(* PLC project Generated.project, CODESYS CODESYS V3.5 SP19 Patch 1 *)
(* stored: creationDateTime 2026-09-14T14:47:22.317175, modificationDateTime 2026-09-14T14:47:22.317175 *)

(* ======================================================================= 🔌 ST_ContactorCheck — Double vérification commande/retour contacteur ─────────────────────────────────────────────────────────────── 🎯 Rôle : Structure de diagnostic pour vérification commande vs retour 📊 Diagnostic : Détection des défauts contacteur (StuckClosed / StuckOpen) 📄 Doc métier : DOC/AF/AF_Partie-03_Contrats_Composants_v2.3.md §2 ======================================================================= *)
TYPE ST_ContactorCheck : STRUCT
  Command : BOOL;  (* Ordre envoyé au contacteur (TRUE = fermé/actif) *)
  Feedback : BOOL;  (* Retour d'état câblé (TRUE = effectivement fermé) *)
  StuckClosed : BOOL;  (* Diag : commande OFF mais retour ON depuis trop longtemps → PowerCutOff *)
  StuckOpen : BOOL;  (* Diag : commande ON mais retour OFF depuis trop longtemps *)
END_STRUCT;
END_TYPE

(* ======================================================================= 🧩 ST_Fault — Brique socle défaut (2 vues : live + latchée) ─────────────────────────────────────────────────────────────── 🎯 Rôle : porter l'état défaut d'un composant, applicable dans TOUS les cas (acquittable ou non), sans brique warning séparée. • Vue LIVE (Error / ErrorId) : suit la cause, retombe seule à 0. • Vue LATCHÉE (Latched / LatchedId): mémorisée au défaut, reste jusqu'au front Reset. Le choix acquittable / non-acquittable se fait PAR CAUSE (ST_FaultCause.Latching), jamais par bloc. 🔒 Sécurité : interlock TOUJOURS sur la cause brute (Error / ErrorId), jamais sur l'acquittement. Reset TOUJOURS effectif, jamais conditionné (std §9). 🧬 Composition : brique de base réutilisable — sortie de FB, struct métier, GVL. Texte IHM NON stocké ici : dérivé côté IHM depuis LatchedId / ErrorId. 📄 Doc : DOC/STDS/CODE_QUALITY_STANDARDS.md §2quinquies / §9 ======================================================================= *)
TYPE ST_Fault : STRUCT
  Error : BOOL;  (* <-- [DIAG] vue LIVE : au moins une cause présente maintenant *)
  ErrorId : WORD;  (* <-- [DIAG] bitfield des causes présentes maintenant (0 si aucune) *)
  Latched : BOOL;  (* <-- [DIAG] vue LATCHÉE : défaut non acquitté, reste jusqu'au front Reset *)
  LatchedId : WORD;  (* <-- [DIAG] ErrorId figé à l'apparition du défaut, effacé au Reset *)
END_STRUCT;
END_TYPE

(* ======================================================================= 🧩 ST_FaultCause — Cause élémentaire alimentant ST_Fault (socle FB_FaultCore) ─────────────────────────────────────────────────────────────── 🎯 Rôle : une cause exprimée EN CLAIR (BOOL + libellé), sans bitfield ni masque. Le FB métier remplit une liste (ARRAY[0..15] OF ST_FaultCause) ; le socle FB_FaultCore en déduit ST_Fault (vue live + vue latchée). 🔒 Sécurité : interlock TOUJOURS sur Active (cause brute), jamais sur le latch. Latching = TRUE → la cause ARME la vue latchée (défaut à acquitter). Latching = FALSE → la cause n'alimente que la vue live (retombe seule). Fail-safe : une cause laissée à Latching=FALSE reste visible en live — pour la rendre acquittable, il faut le déclarer explicitement. 📄 Doc : DOC/STDS/CODE_QUALITY_STANDARDS.md §2quinquies / §9 ======================================================================= *)
TYPE ST_FaultCause : STRUCT
  Active : BOOL;  (* 1 = cause présente maintenant (interlock sur cette valeur) *)
  Latching : BOOL;  (* 1 = cause à acquitter (arme Latched) ; 0 = live seulement *)
  Texte : STRING;  (* libellé prêt IHM (non stocké dans ST_Fault, dérivé côté IHM) *)
END_STRUCT;
END_TYPE

(* ======================================================================= 🪝 ST_fbWinch_Cfg — Configuration statique d'un treuil ─────────────────────────────────────────────────────────────── 🎯 Rôle : Réglages persistants propres à l'instance treuil (statique) 📄 Doc métier : DOC/AF/AF_Partie-10_Fonction_Winch_v2.1.md 📤 Producteur : configuration persistante 📥 Consommateur : FB_Winch (statique uniquement) 🔒 Structs cibles + champs conservés pour garder le décodage %→palier et les deux cadences de rampe DANS FB_Winch (comportement bit-identique). Le champ StepRampDelay est déclaré mais non consommé (usage aval). ======================================================================= *)
TYPE ST_fbWinch_Cfg : STRUCT
  SpeedStepTable : ST_SpeedStepTable;  (* === TABLE DES PALIERS === Table de seuils des paliers de vitesse *)
  DirectionInterlockDelayAscent : TIME := TIME#800ms;  (* === INTERLOCK CHANGEMENT DE SENS === Delai interlock inversion vers montee *)
  DirectionInterlockDelayDescent : TIME := TIME#500ms;  (* Delai interlock inversion vers descente *)
  StepRampDelay : TIME := TIME#700ms;  (* === CADENCE DE RAMPE PALIER === [cible] Tempo de rampe palier (usage aval) *)
  StepRampDelayAscent : TIME := TIME#700ms;  (* [08a] Cadence palier montee (D10, dedie) *)
  StepRampDelayDescent : TIME := TIME#500ms;  (* [08a] Cadence palier descending (D10, dedie) *)
  ContactorFeedbackTimeout : TIME := TIME#500ms;  (* === RETOMBÉE CONTACTEURS === Delai d'attente retombee des contacteurs *)
  SlowdownDistanceTop_M : REAL := 0.5;  (* === RALENTISSEMENT BORDURE === Distance avant limite haute pour ralentir (m) : 0 = arrêt au seuil *)
  SlowdownDistanceBottom_M : REAL := 1;  (* Distance avant limite basse pour ralentir (m) *)
  SlowdownMaxStep : INT := 1;  (* Plafond palier dans zone de ralentissement (1..5) *)
  SpeedStepHystMargin : REAL := 2;  (* === DÉCODAGE %→PALIER (conservé) === [08a] Marge d'hysteresis palier (%) *)
END_STRUCT;
END_TYPE

(* ======================================================================= 🪝 ST_fbWinch_Req — Requête d'axe treuil (producteur PRG_04) ─────────────────────────────────────────────────────────────── 🎯 Rôle : Demande de mouvement, palier et bornes de clamp d'un treuil 📄 Doc métier : DOC/AF/AF_Partie-10_Fonction_Winch_v2.1.md 📤 Producteur : PRG_04_Treuils_Benne (une par treuil M1/M2) 📥 Consommateur : FB_Winch 🔒 Structs cibles + champs conservés pour garder le décodage %→palier et le clamp DANS FB_Winch (comportement bit-identique). SpeedStepReq est consommé par FB_Winch (§5) ; MinStepUp est déclaré mais non consommé (usage aval). ======================================================================= *)
TYPE ST_fbWinch_Req : STRUCT
  RunRequest : BOOL;  (* === ORDRE DE MOUVEMENT === TRUE = mouvement demandé *)
  ReqAscent : BOOL;  (* TRUE = demande montée *)
  ReqDescend : BOOL;  (* TRUE = demande descente *)
  SpeedStepReq : INT;  (* [cible] Palier demandé (1..5, 0 = arrêt) — consommé par FB_Winch *)
  MinStepUp : INT;  (* === BORNES DE CLAMP (agrégées PRG_04) === [cible] Plancher palier montée (usage aval) *)
  MaxStepUp : INT := 5;  (* Plafond palier montée (1..5) *)
  MinStepDown : INT := 0;  (* Plancher palier descente (0 = aucun) -- plongee Kobold *)
  MaxStepDown : INT := 3;  (* Plafond palier descente (1..5) *)
  TopLimitM : REAL := 8.5;  (* === LIMITES EFFECTIVES DU CYCLE === Position limite haute active (m) *)
  BottomLimitM : REAL := -20;  (* Position limite basse active (m) *)
  SyncCoupled : BOOL;  (* === DIAGNOSTIC (jamais lu par la logique FB_Winch) === [diag] Couplage synchro actif (garde de revue) *)
  HomingApproachActive : BOOL;  (* === CHAMPS CONSERVÉS (clamp interne FB_Winch) === [08a] Vitesse limitée au palier 1 (approche homing) *)
END_STRUCT;
END_TYPE

(* ======================================================================= 🪝 ST_fbWinch_Sensors — Mesures et feedbacks d'un treuil ─────────────────────────────────────────────────────────────── 🎯 Rôle : Retours physiques et mesures propres à l'instance treuil 📄 Doc métier : DOC/AF/AF_Partie-10_Fonction_Winch_v2.1.md 📤 Producteur : PRG_04_Treuils_Benne / acquisition 📥 Consommateur : FB_Winch 🔒 Structs cibles + champs conservés pour garder le garde-fou vitesse DANS FB_Winch (comportement bit-identique). Les champs MeasuredSpeedMps / MeasuredSpeedValid sont déclarés mais non consommés (usage aval). ======================================================================= *)
TYPE ST_fbWinch_Sensors : STRUCT
  CablePosM : REAL;  (* === POSITION ET RÉFÉRENCEMENT === Position actuelle du cable (m) *)
  Homed : BOOL;  (* Statut treuil reference *)
  HomingSuspect : BOOL;  (* Incertitude / doute sur le referencement *)
  ContactorsAllOff : BOOL;  (* === RETOURS CONTACTEURS === TRUE = relais sens + C1..C4 tous retombés (ex-FwdRevSpeedFeedbackOff) *)
  MeasuredSpeedMps : REAL;  (* === MESURE VITESSE === [cible] Mesure vitesse réelle (m/s) — usage aval *)
  MeasuredSpeedValid : BOOL;  (* [cible] Mesure exploitable — usage aval *)
  MeasuredSpeedBand : INT := 0;  (* [08a] Bande vitesse réelle validée (garde-fou conservé dans FB_Winch) *)
  SpeedGuardEnable : BOOL := TRUE;  (* === GARDE-FOU VITESSE (conservé) === [08a] Activation garde-fou changement de palier *)
  SpeedGuardReady : BOOL := FALSE;  (* [08a] Conditions de stabilité validées *)
END_STRUCT;
END_TYPE

(* ======================================================================= 🪜 ST_SpeedStepTable — Table des paliers de vitesse contacteurs ─────────────────────────────────────────────────────────────── 🎯 Rôle : Structure de configuration des contacteurs et seuils par palier 📄 Doc métier : DOC/AF/AF_Partie-10_Fonction_Winch_v2.1.md ======================================================================= *)
TYPE ST_SpeedStepTable : STRUCT
  P1R1 : BOOL;  (* === PALIER 1 (VITESSE MINIMALE) === Contacteur 1 pour Palier 1 *)
  P1R2 : BOOL;  (* Contacteur 2 pour Palier 1 *)
  P1R3 : BOOL;  (* Contacteur 3 pour Palier 1 *)
  P1R4 : BOOL;  (* Contacteur 4 pour Palier 1 *)
  P2R1 : BOOL;  (* === PALIER 2 === Contacteur 1 pour Palier 2 *)
  P2R2 : BOOL;  (* Contacteur 2 pour Palier 2 *)
  P2R3 : BOOL;  (* Contacteur 3 pour Palier 2 *)
  P2R4 : BOOL;  (* Contacteur 4 pour Palier 2 *)
  P3R1 : BOOL;  (* === PALIER 3 === Contacteur 1 pour Palier 3 *)
  P3R2 : BOOL;  (* Contacteur 2 pour Palier 3 *)
  P3R3 : BOOL;  (* Contacteur 3 pour Palier 3 *)
  P3R4 : BOOL;  (* Contacteur 4 pour Palier 3 *)
  P4R1 : BOOL;  (* === PALIER 4 === Contacteur 1 pour Palier 4 *)
  P4R2 : BOOL;  (* Contacteur 2 pour Palier 4 *)
  P4R3 : BOOL;  (* Contacteur 3 pour Palier 4 *)
  P4R4 : BOOL;  (* Contacteur 4 pour Palier 4 *)
  P5R1 : BOOL;  (* === PALIER 5 (VITESSE MAXIMALE) === Contacteur 1 pour Palier 5 *)
  P5R2 : BOOL;  (* Contacteur 2 pour Palier 5 *)
  P5R3 : BOOL;  (* Contacteur 3 pour Palier 5 *)
  P5R4 : BOOL;  (* Contacteur 4 pour Palier 5 *)
  StepThreshold_Pct : ARRAY[1..5] OF REAL;  (* === SEUILS DE TRANSITION (%) === Seuils de changement de palier (0..100%) *)
END_STRUCT;
END_TYPE

(* ======================================================================= 🪝 FB_Winch — Directeur d'un treuil individuel (M1 / M2) ─────────────────────────────────────────────────────────────── 🎯 Rôle : Pilotage d'un treuil individuel (contacteurs de sens et de vitesse) 📄 Doc métier : DOC/AF/AF_Partie-10_Fonction_Winch_v2.1.md 🔌 Interface : FB de mouvement (Enable, SafeStop, RunRequest via WinchRequest) 🔒 Sécurité : Interlock inversion de sens et gestion des autorisations 🔧 Interface plate → structs (WinchRequest / Sensors / Config), logique interne conservée (comportement bit-identique). ======================================================================= *)
FUNCTION_BLOCK FB_Winch
  VAR_INPUT
    Enable : BOOL;  (* === COMMANDES ET CONSIGNES === --> [CMD] Autorisation generale FB (TRUE=Autorise) *)
    Reset : BOOL;  (* --> [CMD] Acquittement defaut (front) *)
    PowerContactorEngaged : BOOL;  (* --> [SAFE] Statut contacteur de ligne / puissance *)
    WinchRequest : ST_fbWinch_Req;  (* === REQUÊTE D'AXE (struct) === --> [REQ] RunRequest + 2 bits de sens, palier et limites *)
    Sensors : ST_fbWinch_Sensors;  (* === MESURES ET FEEDBACKS (struct) === --> [HW] Position, referencement, contacteurs, vitesse *)
    Config : ST_fbWinch_Cfg;  (* === CONFIGURATION STATIQUE (struct) === --> [CFG] Table paliers, delais, ralentissement *)
    SafeStop : BOOL;  (* === SECOURS ET PERMIS DE SÉCURITÉ === --> [SAFE] Arret rapide de securite *)
    DescendPermit : BOOL := FALSE;  (* --> [SAFE] Permis de descente (mou de cable) *)
    AscentPermit : BOOL := FALSE;  (* --> [SAFE] Permis de montee (fin de course haut) *)
    BypassContactorCheck : BOOL;  (* === BYPASSES ET SIMULATION === --> [TST] Bypass diagnostic contacteurs (simu) *)
    BypassGlobal : BOOL;  (* --> [TST] Force ErrorId=0, ignore erreurs *)
  END_VAR
  VAR_OUTPUT
    Ready : BOOL;  (* === ETATS IEC ET SYNOPTIQUE === <-- [STAT] FB pret a fonctionner *)
    Fault : ST_Fault;  (* 🧩 Statut transverse (forme cible ST_Fault) *)
    RelayFwd : BOOL;  (* === ORDRES ACTIONNEURS (CONTACTEURS) === <-- [ACT] Ordre contacteur sens montee *)
    RelayRev : BOOL;  (* <-- [ACT] Ordre contacteur sens descente *)
    Contactor1 : BOOL;  (* <-- [ACT] Ordre contacteur vitesse palier 1 *)
    Contactor2 : BOOL;  (* <-- [ACT] Ordre contacteur vitesse palier 2 *)
    Contactor3 : BOOL;  (* <-- [ACT] Ordre contacteur vitesse palier 3 *)
    Contactor4 : BOOL;  (* <-- [ACT] Ordre contacteur vitesse palier 4 *)
    RequestedStep : INT;  (* === DIAGNOSTICS ET MESURES === <-- [DIAG] Palier brut calcule par SpeedStep *)
    StepNumber : INT;  (* <-- [DIAG] Palier metier temporise actif *)
    BusinessStepDelayElapsed : TIME;  (* <-- [DIAG] Ecoule tempo metier palier *)
    SpeedGuardLimited : BOOL;  (* <-- [DIAG] Statut limitation par garde-fou *)
    ContactorsCheck : ST_ContactorCheck;  (* <-- [DIAG] Diagnostic concorde contacteurs *)
    InTopSlowdownZone : BOOL;  (* <-- [DIAG] Zone de ralentissement haut active *)
    InBottomSlowdownZone : BOOL;  (* <-- [DIAG] Zone de ralentissement bas active *)
    CommandedAscent : BOOL;  (* <-- [DIAG] Sens interne mémorisé : montée *)
    CommandedDescend : BOOL;  (* <-- [DIAG] Sens interne mémorisé : descente *)
    RequestConflict : BOOL;  (* <-- [DIAG] Double demande de sens détectée *)
    DirectionChangeDelayElapsed : TIME;  (* <-- [DIAG] Ecoule delai changement de sens *)
    DirectionChangePending : BOOL;  (* <-- [DIAG] Changement de sens en attente *)
    SenseHoldRequest : BOOL;  (* === INTENTION DE MAINTIEN DU CONTACTEUR DE SENS (§3bis) === <-- [ACT] Demande a la barriere finale de TENIR le contacteur de sens apres chute de palier a 0 (inertie moteur), bornee par T_hold_internal *)
  END_VAR
  VAR
    SpeedStep : FB_SpeedStep;  (* === SOUS-INSTANCES FB === * [INST] Decodage paliers vitesse *)
    DirectionInterlock : FB_WinchDirectionInterlock;  (* * [INST] Interlock changement de sens (D18) *)
    StepShaper : FB_WinchStepShaper;  (* * [INST] Cadencement de palier (D10) *)
    ResetEdge : R_TRIG;  (* === DETECTEURS ET TIMERS INTERNES === . [LOC] Detecteur front montant Reset *)
    EnableRisingEdge : R_TRIG;  (* . [LOC] Detecteur front montant Enable (D18) *)
    TonContactorsDropped : TON;  (* . [LOC] Temporisation retombee contacteurs *)
    AllContactorsCommandedOff : BOOL;  (* === VARIABLES LOCALES CALCULÉES === . [LOC] Tous contacteurs commandes a FALSE *)
    RampTargetStep : INT;  (* . [LOC] Palier demandé par l'arbitrage amont *)
    EffectiveSafeStop : BOOL;  (* . [LOC] SafeStop effectif incluant permis *)
    DirectionConflict : BOOL;  (* . [LOC] Les deux demandes de sens sont actives *)
    ActiveMaxStep : INT;  (* . [LOC] Plafond palier actif dynamique *)
    EffectiveStepRampDelay : TIME;  (* . [LOC] Cadence palier selon sens, distincte interlock *)
    SenseHoldTimer : TON;  (* === MAINTIEN DU CONTACTEUR DE SENS (§3bis) === . [LOC] Garde interne T_hold_internal (< MaxSenseHoldTime barriere) *)
    SenseHoldActiveInt : BOOL;  (* . [LOC] Maintien de sens interne en cours *)
    PrevStepNumber : INT;  (* . [LOC] Palier temporise du scan precedent (detection chute a 0) *)
    SenseHoldHardCut : BOOL;  (* . [LOC] Coupure dure active (interdit tout maintien) *)
    SpeedStepConfigFaultLatched : BOOL;  (* Latches défauts *)
    instFault : FB_FaultCore;  (* Socle défaut * [INST] Socle défaut transverse *)
    instCauses : ARRAY[0..15] OF ST_FaultCause;  (* . [LOC] Table des causes nommées *)
  END_VAR

            

// === IMPLEMENTATION ===

{region "§1 Causes & Socle Défaut (évalué en continu)"}
// 🔑 1. FRONTS & REARMEMENT
ResetEdge(CLK := Reset);
EnableRisingEdge(CLK := Enable);

IF ResetEdge.Q OR BypassGlobal THEN
    SpeedStepConfigFaultLatched := FALSE;
    ContactorsCheck.StuckClosed := FALSE;
END_IF;

IF Enable AND SpeedStep.ConfigError THEN
    SpeedStepConfigFaultLatched := TRUE;
END_IF;

// FB_Safety_Winch est l'unique proprietaire de la detection contacteur colle.
// FB_Winch conserve le champ public pour compatibilite IHM/Troubleshooting,
// mais ne produit plus ce defaut.
instCauses[1].Active   := FALSE;
instCauses[1].Latching := TRUE;
instCauses[1].Texte    := 'Contacteur colle gere par FB_Safety_Winch ';

instCauses[2].Active   := SpeedStepConfigFaultLatched;
instCauses[2].Latching := TRUE;
instCauses[2].Texte    := 'Configuration table des paliers vitesse invalide';

// Appel du socle de défaut
instFault(Enable := Enable, Reset := Reset, Causes := instCauses);
Fault := instFault.Fault;
{endregion}

{region "§2 Gate neutralisation"}
// 🛑 2. GATE
IF NOT Enable THEN
    SpeedStep(Enable := FALSE, SpeedStepReq := 0, Table := Config.SpeedStepTable);
    DirectionInterlock(Enable := FALSE, EnableRising := FALSE, Reset := Reset, ReqAscent := FALSE, ReqDescend := FALSE,
                       ChangeDelayAscent := Config.DirectionInterlockDelayAscent,
                       ChangeDelayDescent := Config.DirectionInterlockDelayDescent);
    StepShaper(Enable := FALSE, TargetStep := 0, StepRampDelay := Config.StepRampDelayAscent);
    RelayFwd := FALSE;
    RelayRev := FALSE;
    Contactor1 := FALSE; Contactor2 := FALSE; Contactor3 := FALSE; Contactor4 := FALSE;
    RequestedStep := 0;
    StepNumber := StepShaper.ShapedStep;
    CommandedAscent := DirectionInterlock.CommandedAscent;
    CommandedDescend := DirectionInterlock.CommandedDescend;
    RequestConflict := DirectionInterlock.RequestConflict;
    DirectionChangePending := DirectionInterlock.DirectionChangePending;
    TonContactorsDropped(IN := FALSE);
    ContactorsCheck.Command := FALSE;
    ContactorsCheck.Feedback := NOT Sensors.ContactorsAllOff;
    InTopSlowdownZone := FALSE;
    InBottomSlowdownZone := FALSE;
    // §3bis : coupure dure -> aucun maintien de sens possible, etat interne purge.
    SenseHoldRequest := FALSE;
    SenseHoldActiveInt := FALSE;
    SenseHoldTimer(IN := FALSE, PT := T#900ms);
    PrevStepNumber := 0;
    Ready := FALSE;
    RETURN;
END_IF;

Ready := Enable AND NOT Fault.Latched;
{endregion}

{region "§3 Permis et zones de ralentissement"}
DirectionConflict := WinchRequest.ReqAscent AND WinchRequest.ReqDescend;
EffectiveSafeStop := SafeStop OR DirectionConflict
                     OR (WinchRequest.ReqAscent AND NOT AscentPermit)
                     OR (WinchRequest.ReqDescend AND NOT DescendPermit);

InTopSlowdownZone := Sensors.Homed AND NOT Sensors.HomingSuspect AND (Sensors.CablePosM >= (WinchRequest.TopLimitM - Config.SlowdownDistanceTop_M));
InBottomSlowdownZone := Sensors.Homed AND NOT Sensors.HomingSuspect AND (Sensors.CablePosM <= (WinchRequest.BottomLimitM + Config.SlowdownDistanceBottom_M));

IF WinchRequest.ReqAscent AND NOT WinchRequest.ReqDescend THEN
    ActiveMaxStep := WinchRequest.MaxStepUp;
    IF InTopSlowdownZone THEN
        ActiveMaxStep := MIN(ActiveMaxStep, Config.SlowdownMaxStep);
    END_IF;
ELSIF WinchRequest.ReqDescend AND NOT WinchRequest.ReqAscent THEN
    ActiveMaxStep := WinchRequest.MaxStepDown;
    IF InBottomSlowdownZone THEN
        ActiveMaxStep := MIN(ActiveMaxStep, Config.SlowdownMaxStep);
    END_IF;
ELSE
    ActiveMaxStep := WinchRequest.MaxStepUp;
END_IF;

IF WinchRequest.HomingApproachActive THEN
    ActiveMaxStep := 1;
END_IF;
{endregion}

{region "§4 Interlock direction"}
// 🔀 4. INTERLOCK DIRECTION (extrait dans FB_WinchDirectionInterlock, D18)
DirectionInterlock(
    Enable := (StepNumber = 0) AND Sensors.ContactorsAllOff,
    EnableRising := EnableRisingEdge.Q,
    Reset := Reset,
    ReqAscent := WinchRequest.ReqAscent,
    ReqDescend := WinchRequest.ReqDescend,
    ChangeDelayAscent := Config.DirectionInterlockDelayAscent,
    ChangeDelayDescent := Config.DirectionInterlockDelayDescent
);
CommandedAscent := DirectionInterlock.CommandedAscent;
CommandedDescend := DirectionInterlock.CommandedDescend;
RequestConflict := DirectionInterlock.RequestConflict;
DirectionChangePending := DirectionInterlock.DirectionChangePending;
DirectionChangeDelayElapsed := DirectionInterlock.DelayElapsed;
{endregion}

{region "§5 Paliers vitesse et contacteurs"}
// -B : la consigne est désormais un PALIER discret (WinchRequest.SpeedStepReq,
// 1..5, 0 = arrêt) produit par l'arbitrage. Plus de décodage %→palier ici.
IF DirectionChangePending OR NOT (WinchRequest.ReqAscent OR WinchRequest.ReqDescend) OR EffectiveSafeStop OR NOT WinchRequest.RunRequest THEN
    RampTargetStep := 0;
ELSE
    RampTargetStep := WinchRequest.SpeedStepReq;
END_IF;

SpeedStep(
    Enable := (RampTargetStep > 0),
    SpeedStepReq := RampTargetStep,
    Table := Config.SpeedStepTable,
    MaxStepNumber := ActiveMaxStep
);
RequestedStep := SpeedStep.StepNumber;

// 🛡️ Garde-fou vitesse : bride le palier demande si la vitesse n'est pas stable
// (SpeedGuardReady=FALSE -> palier 1) ou si la bande mesuree est inferieure au
// palier demande (pas de passage aux paliers superieurs sans vitesse confirmee).
SpeedGuardLimited := FALSE;
IF Sensors.SpeedGuardEnable THEN
    IF NOT Sensors.SpeedGuardReady THEN
        IF RequestedStep > 1 THEN
            RequestedStep := 1;
            SpeedGuardLimited := TRUE;
        END_IF;
    ELSIF (Sensors.MeasuredSpeedBand >= 1) AND (Sensors.MeasuredSpeedBand <= 5) AND (RequestedStep > Sensors.MeasuredSpeedBand) THEN
        RequestedStep := Sensors.MeasuredSpeedBand;
        SpeedGuardLimited := TRUE;
    END_IF;
END_IF;

// 🤿 Plancher palier descente -- plongee Kobold.
// Injecte MinStepDown sur la CIBLE (RequestedStep, consommee par le shaper ci-dessous),
// JAMAIS sur StepNumber directement. Actif uniquement en descente commandee
// ET NON bloquee par un arret/permis (NOT EffectiveSafeStop) : un permis descente FALSE
// doit interdire physiquement le mouvement, sans re-atterrissage du plancher.
// Le sens doit aussi etre deja adopte : pendant DirectionChangePending, le
// StepNumber doit rester a 0 afin que le temps mort d'inversion puisse s'ecouler.
// (RunRequest AND ReqDescend) : relache joystick (RunRequest=FALSE) -> aucun plancher,
// l'arret franc RequestedStep=0 / RampTargetStep=0 est preserve.
// Regle d'agregation : le PLAFOND GAGNE -- si le plancher depasse le plafond courant
// ActiveMaxStep (ex. SlowdownMaxStep -> palier 1 en bordure basse), on borne au plafond.
IF WinchRequest.RunRequest AND WinchRequest.ReqDescend AND NOT WinchRequest.ReqAscent
   AND (WinchRequest.MinStepDown > 0) AND NOT EffectiveSafeStop
   AND NOT DirectionChangePending AND CommandedDescend THEN
    IF RequestedStep < WinchRequest.MinStepDown THEN
        RequestedStep := WinchRequest.MinStepDown;
    END_IF;
    IF RequestedStep > ActiveMaxStep THEN
        RequestedStep := ActiveMaxStep;
    END_IF;
END_IF;

// ⚙️ Cadencement de palier (extrait dans FB_WinchStepShaper, D10).
// Les deux cadences historiques sont preservees sans reutiliser les delais
// d'interlock direction : 1 s en montee, 500 ms en descente.
IF CommandedDescend THEN
    EffectiveStepRampDelay := Config.StepRampDelayDescent;
ELSE
    EffectiveStepRampDelay := Config.StepRampDelayAscent;
END_IF;
StepShaper(
    Enable := Enable,
    TargetStep := RequestedStep,
    StepRampDelay := EffectiveStepRampDelay
);
StepNumber := StepShaper.ShapedStep;
BusinessStepDelayElapsed := StepShaper.StepDelayElapsed;

IF StepNumber > 0 AND CommandedAscent THEN
    RelayFwd := TRUE;
    RelayRev := FALSE;
ELSIF StepNumber > 0 AND CommandedDescend THEN
    RelayFwd := FALSE;
    RelayRev := TRUE;
ELSE
    RelayFwd := FALSE;
    RelayRev := FALSE;
END_IF;

// 🛡️ FIX contacteurs (audit CONTACTEURS_2026-08-31) + SOLUTION : ré-émettre les
// contacteurs depuis FB_SpeedStep (décodage TABLE ST_SpeedStepTable cumulatif :
// P1=0, P2={K1}, P3={K1,K2}, P4={K1,K2,K3}, P5={K1,K2,K3,K4}) sur le palier SHAPÉ,
// au lieu de l'ancien décodage one-hot exclusif (ContactorN := StepNumber=N) qui
// éteignait les paliers inférieurs et ne couvrait pas le palier 5.
SpeedStep(
    Enable          := (StepNumber > 0),
    SpeedStepReq    := StepNumber,
    Table           := Config.SpeedStepTable,
    MaxStepNumber   := ActiveMaxStep
);
Contactor1 := SpeedStep.Contactor1;
Contactor2 := SpeedStep.Contactor2;
Contactor3 := SpeedStep.Contactor3;
Contactor4 := SpeedStep.Contactor4;

AllContactorsCommandedOff := (NOT RelayFwd) AND (NOT RelayRev)
                             AND (NOT Contactor1) AND (NOT Contactor2) AND (NOT Contactor3) AND (NOT Contactor4);

ContactorsCheck.Command  := NOT AllContactorsCommandedOff;
ContactorsCheck.Feedback := NOT Sensors.ContactorsAllOff;
TonContactorsDropped(IN := FALSE, PT := Config.ContactorFeedbackTimeout);
ContactorsCheck.StuckClosed := FALSE; // force a FALSE (Phase 0) : detection contacteur colle produite par FB_Safety_Winch, re-alimentee a la phase suivante
ContactorsCheck.StuckOpen := FALSE;

IF Fault.Error THEN
    RelayFwd := FALSE;
    RelayRev := FALSE;
    Contactor1 := FALSE; Contactor2 := FALSE; Contactor3 := FALSE; Contactor4 := FALSE;
END_IF;
{endregion}

{region "§5bis Intention de maintien du contacteur de sens (§3bis)"}
// Quand le palier temporise StepNumber vient de retomber a 0 alors qu'un sens etait
// commande, FB_Winch DEMANDE a la barriere finale (FB_WinchOutputInterlock) de TENIR
// le contacteur de sens le temps que le moteur ralentisse (inertie). Borne par
// T_hold_internal (garde interne, < MaxSenseHoldTime de la barriere = T#1s).
// Coupures dures -> retombee immediate, jamais de maintien (SafeStop / defaut / perte
// puissance / NOT Enable geree a la gate §2).
SenseHoldHardCut := (NOT PowerContactorEngaged) OR EffectiveSafeStop OR Fault.Error;

IF SenseHoldHardCut THEN
    SenseHoldActiveInt := FALSE;
ELSIF (PrevStepNumber > 0) AND (StepNumber = 0) AND (CommandedAscent OR CommandedDescend) THEN
    SenseHoldActiveInt := TRUE;   // front de chute de palier a 0 avec sens encore actif
END_IF;

// Maintien interne aligné sur MaxSenseHoldTime de FB_WinchOutputInterlock (T#400ms).
SenseHoldTimer(IN := SenseHoldActiveInt, PT := T#400ms);
IF SenseHoldTimer.Q OR (StepNumber > 0) THEN
    SenseHoldActiveInt := FALSE;  // borne de temps atteinte, ou nouveau mouvement demande
END_IF;

SenseHoldRequest := SenseHoldActiveInt AND NOT SenseHoldHardCut;
PrevStepNumber := StepNumber;
{endregion}

          
END_FUNCTION_BLOCK

(* ======================================================================= 🧩 FB_FaultCore — Socle de remplissage de ST_Fault (vue live + vue latchée) ─────────────────────────────────────────────────────────────── 🎯 Rôle : à partir d'une LISTE de causes en clair (ARRAY[0..15] OF ST_FaultCause), produire la brique ST_Fault : • Error / ErrorId : vue LIVE, suit les causes Active, retombe seule. • Latched / LatchedId: vue LATCHÉE, chaque bit figé à l'apparition d'une cause `Active AND Latching`, conservé jusqu'au front Reset. 🔒 Sécurité : - interlock TOUJOURS sur `Causes[i].Active` (cause brute), jamais sur le latch. - Reset TOUJOURS effectif, jamais conditionné (std §9) — agit même Enable=FALSE. - Latching=FALSE → cause visible en LIVE seulement (fail-safe : reste visible). - un défaut laté non acquitté reste publié même FB désactivé (pas d'effacement silencieux sur bascule Enable OFF→ON sans Reset). - une cause à acquitter réapparue re-arme son bit (ré-alarme). 🧬 Un seul socle, réutilisé par tout FB `standard` qui expose un ST_Fault. Pas de State, pas de Warning, pas de texte — hors périmètre de ce socle. 📄 Doc : DOC/STDS/CODE_QUALITY_STANDARDS.md §2quinquies / §9 ======================================================================= *)
FUNCTION_BLOCK FB_FaultCore
  VAR_INPUT
    Enable : BOOL;  (* --> [CMD] Autorisation générale du FB porteur *)
    Reset : BOOL;  (* --> [CMD] Front d'acquittement (jamais conditionné, §9) *)
    Causes : ARRAY[0..15] OF ST_FaultCause;  (* --> [CMD] Liste des causes en clair (Active / Latching / Texte) *)
  END_VAR
  VAR_OUTPUT
    Ready : BOOL;  (* <-- [STAT] FB porteur autorisé (= Enable) *)
    Fault : ST_Fault;  (* <-- [DIAG] Brique défaut (mappée 1:1 sur la sortie du FB porteur) *)
  END_VAR
  VAR
    ResetEdge : R_TRIG;  (* . [LOC] Front montant Reset *)
    Latch : ARRAY[0..15] OF BOOL;  (* . [LOC] Bit laté par cause, jusqu'au Reset *)
    i : INT;  (* . [LOC] Index de parcours de la liste *)
  END_VAR

            

{region "§1 Reset (front, toujours effectif)"}
// Front Reset : efface tous les latches. Jamais conditionné, agit même Enable=FALSE (§9).
Ready := Enable;
ResetEdge(CLK := Reset);
IF ResetEdge.Q THEN
    FOR i := 0 TO 15 DO Latch[i] := FALSE; END_FOR;
END_IF;
{endregion}

{region "§2 Vue LIVE — Error / ErrorId"}
// Bitfield des causes présentes MAINTENANT. Retombe seule à 0 quand les causes disparaissent.
// Non évaluée si Enable=FALSE (pas de lecture de cause hors autorisation).
Fault.ErrorId := 0;
IF Enable THEN
    FOR i := 0 TO 15 DO
        IF Causes[i].Active THEN
            Fault.ErrorId := Fault.ErrorId OR SHL(WORD#1, INT_TO_DWORD(i));
        END_IF;
    END_FOR;
END_IF;
Fault.Error := (Fault.ErrorId <> 0);
{endregion}

{region "§3 Armement des latches (causes à acquitter)"}
// Une cause Active ET Latching arme son bit ; le bit reste jusqu'au front Reset (§1),
// même si la cause disparaît. Réapparition => ré-armement (ré-alarme).
IF Enable THEN
    FOR i := 0 TO 15 DO
        IF Causes[i].Active AND Causes[i].Latching THEN
            Latch[i] := TRUE;
        END_IF;
    END_FOR;
END_IF;
{endregion}

{region "§4 Vue LATCHÉE — Latched / LatchedId"}
// Toujours publiée, y compris Enable=FALSE : un défaut non acquitté reste visible.
Fault.LatchedId := 0;
FOR i := 0 TO 15 DO
    IF Latch[i] THEN
        Fault.LatchedId := Fault.LatchedId OR SHL(WORD#1, INT_TO_DWORD(i));
    END_IF;
END_FOR;
Fault.Latched := (Fault.LatchedId <> 0);
{endregion}

          
END_FUNCTION_BLOCK

(* ======================================================================= FB_SpeedStep — Décodeur palier vers contacteurs Rôle : applique les bornes de palier puis lit la table contacteurs. Le calcul de la consigne discrète est fait par le producteur amont. ======================================================================= *)
FUNCTION_BLOCK FB_SpeedStep
  VAR_INPUT
    Enable : BOOL;
    SpeedStepReq : INT := 0;  (* --> [CMD] Palier demandé (0..5) *)
    Table : ST_SpeedStepTable;  (* --> [CFG] Table contacteurs propre au treuil *)
    MinStepNumber : INT := 1;  (* --> [CFG] Plancher palier, rétro-compatible *)
    MaxStepNumber : INT := 5;  (* --> [CFG] Plafond palier atteignable *)
  END_VAR
  VAR_OUTPUT
    StepNumber : INT;  (* <-- [STAT] Palier actif (0..5) *)
    Contactor1 : BOOL;  (* <-- [ACT] Ordre contacteur vitesse palier 1 *)
    Contactor2 : BOOL;  (* <-- [ACT] Ordre contacteur vitesse palier 2 *)
    Contactor3 : BOOL;  (* <-- [ACT] Ordre contacteur vitesse palier 3 *)
    Contactor4 : BOOL;  (* <-- [ACT] Ordre contacteur vitesse palier 4 *)
    ConfigError : BOOL;  (* <-- [DIAG] Table de paliers invalide *)
    ConfigErrorId : WORD;  (* <-- [DIAG] Bitfield erreur table *)
  END_VAR
  VAR
    _ConfigValid : BOOL;
    _ConfigErrorIdInt : WORD;
    _MaxStepClamped : INT;
    _MinStepClamped : INT;
  END_VAR

            

{region "§0 Bornes et validation table"}
// Le plafond est borné avant le plancher : si le plancher demandé dépasse le
// plafond de sécurité, celui-ci garde la priorité.
_MaxStepClamped := LIMIT(1, MaxStepNumber, 5);
_MinStepClamped := LIMIT(1, MinStepNumber, _MaxStepClamped);

// Les seuils restent validés pour conserver le diagnostic table historique.
// Ils ne participent plus au calcul du palier dans ce FB.
_ConfigValid := TRUE;
_ConfigErrorIdInt := 16#0000;
IF NOT (Table.StepThreshold_Pct[1] < Table.StepThreshold_Pct[2] AND
        Table.StepThreshold_Pct[2] < Table.StepThreshold_Pct[3] AND
        Table.StepThreshold_Pct[3] < Table.StepThreshold_Pct[4] AND
        Table.StepThreshold_Pct[4] < Table.StepThreshold_Pct[5]) THEN
    _ConfigValid := FALSE;
    _ConfigErrorIdInt := _ConfigErrorIdInt OR 16#0001;
END_IF;
IF (Table.StepThreshold_Pct[1] < 0.0) OR (Table.StepThreshold_Pct[5] > 100.0) THEN
    _ConfigValid := FALSE;
    _ConfigErrorIdInt := _ConfigErrorIdInt OR 16#0001;
END_IF;
ConfigErrorId := _ConfigErrorIdInt;
ConfigError := (ConfigErrorId <> 16#0000);
{endregion}

{region "§1 Gate"}
// Relâche ou table invalide : aucun plancher ne peut maintenir un contacteur.
IF (NOT Enable) OR (NOT _ConfigValid) OR (SpeedStepReq <= 0) THEN
    StepNumber := 0;
    Contactor1 := FALSE; Contactor2 := FALSE; Contactor3 := FALSE; Contactor4 := FALSE;
    RETURN;
END_IF;
{endregion}

{region "§2 Clamp et table contacteurs"}
// Le plancher agit sur la cible. StepNumber ne reçoit jamais directement
// MinStepNumber ; LIMIT final garantit la plage 1..5 après le plafond.
StepNumber := LIMIT(_MinStepClamped, SpeedStepReq, _MaxStepClamped);

CASE StepNumber OF
    1:  Contactor1 := Table.P1R1; Contactor2 := Table.P1R2; Contactor3 := Table.P1R3; Contactor4 := Table.P1R4;
    2:  Contactor1 := Table.P2R1; Contactor2 := Table.P2R2; Contactor3 := Table.P2R3; Contactor4 := Table.P2R4;
    3:  Contactor1 := Table.P3R1; Contactor2 := Table.P3R2; Contactor3 := Table.P3R3; Contactor4 := Table.P3R4;
    4:  Contactor1 := Table.P4R1; Contactor2 := Table.P4R2; Contactor3 := Table.P4R3; Contactor4 := Table.P4R4;
    5:  Contactor1 := Table.P5R1; Contactor2 := Table.P5R2; Contactor3 := Table.P5R3; Contactor4 := Table.P5R4;
ELSE
    // Défense en profondeur face à une divergence type/outil.
    StepNumber := 0;
    Contactor1 := FALSE; Contactor2 := FALSE; Contactor3 := FALSE; Contactor4 := FALSE;
END_CASE;
{endregion}

          
END_FUNCTION_BLOCK

(* ======================================================================= 🔀 FB_WinchDirectionInterlock — Interlock de changement de sens ─────────────────────────────────────────────────────────────── 🎯 Rôle : Temporise l'INVERSION de sens d'un treuil, en creditant le temps d'arret physique reel deja ecoule (dead time) 📄 Doc métier : DOC/AF/AF_Partie-10_Fonction_Winch_v2.1.md 🔌 Interface : Brique technique (contrat light, pas de defaut) 🔒 Sécurité : D18 — au front montant Enable, n'adopte pas le sens immediatement (temps mort) ; pas de redemarrage inrush. Le sens IDENTIQUE au dernier sens adopte reste toujours immediat depuis le neutre : seule l'INVERSION est temporisee. Purge de DeadTimeArmed garantie des que le temps mort est ecoule (T325 phase 1). Limite residuelle connue (T325 phase 2, non couverte ici) : si la demande redevient le MEME sens que le dernier commande alors que DeadTimeArmed vient d'etre arme, DirectionChanged reste FALSE et le temps mort ne peut jamais etre mesure -- seule sortie encore possible dans ce cas precis : retour au neutre ou Reset. ======================================================================= *)
FUNCTION_BLOCK FB_WinchDirectionInterlock
  VAR_INPUT
    Enable : BOOL;  (* --> [CMD] Gate TON (TRUE = treuil arrete, contacteurs retombes) *)
    EnableRising : BOOL;  (* --> [CMD] Front montant Enable du FB parent (D18) *)
    Reset : BOOL;  (* --> [CMD] Acquittement defaut (front) : purge la memoire de direction *)
    ReqAscent : BOOL;  (* --> [CMD] Demande montée *)
    ReqDescend : BOOL;  (* --> [CMD] Demande descente *)
    ChangeDelayAscent : TIME;  (* --> [CFG] Delai interlock changement de sens montee *)
    ChangeDelayDescent : TIME;  (* --> [CFG] Delai interlock changement de sens descente *)
  END_VAR
  VAR_OUTPUT
    CommandedAscent : BOOL;  (* <-- [DIAG] Sens interne mémorisé : montée *)
    CommandedDescend : BOOL;  (* <-- [DIAG] Sens interne mémorisé : descente *)
    RequestConflict : BOOL;  (* <-- [DIAG] Double demande refusée *)
    DirectionChangePending : BOOL;  (* <-- [DIAG] Changement de sens en attente *)
    DelayElapsed : TIME;  (* <-- [DIAG] Ecoule delai changement de sens *)
  END_VAR
  VAR
    DirectionChangeDelay : TON;  (* . [LOC] Xa->Xb : compte le reliquat apres la nouvelle demande d'inversion *)
    StoppedTimer : TON;  (* . [LOC] Xc->Xd : accumule le temps d'arret physique reel (Enable, hors demande) *)
    CapturedStoppedTime : TIME;  (* . [LOC] Arret reel credite, fige au front RequestActive, purge une fois consomme *)
    RemainingDelay : TIME;  (* . [LOC] Reliquat a appliquer par DirectionChangeDelay (delai plein - arret credite) *)
    EffectiveDelay : TIME;  (* . [LOC] Delai plein selon sens demande *)
    MaxDirectionDelay : TIME;  (* . [LOC] MAX(ChangeDelayAscent, ChangeDelayDescent) : base d'accumulation StoppedTimer *)
    DeadTimeArmed : BOOL;  (* . [LOC] Temps mort D18 arme (front Enable) *)
    LastAscent : BOOL;  (* . [LOC] Dernier sens adopté : montée *)
    LastDescend : BOOL;  (* . [LOC] Dernier sens adopté : descente *)
    RequestActive : BOOL;  (* . [LOC] Une seule demande de sens active *)
    RequestActiveRising : R_TRIG;  (* . [LOC] Front nouvelle demande : capture le credit avant le rappel de StoppedTimer *)
    DirectionChanged : BOOL;  (* . [LOC] Demande différente du sens commandé *)
    ResetEdge : R_TRIG;  (* . [LOC] Front Reset : purge la memoire de direction *)
  END_VAR

            

// === IMPLEMENTATION ===

// Front Reset : purge la memoire de direction (un acquittement conscient reinitialise
// l'historique, une reprise apres Reset est un depart propre, pas une inversion).
ResetEdge(CLK := Reset);
IF ResetEdge.Q THEN
    LastAscent := FALSE;
    LastDescend := FALSE;
    CommandedAscent := FALSE;
    CommandedDescend := FALSE;
    DeadTimeArmed := FALSE;
    DirectionChangePending := FALSE;
    CapturedStoppedTime := T#0ms;
END_IF;

RequestConflict := ReqAscent AND ReqDescend;
RequestActive := (ReqAscent OR ReqDescend) AND NOT RequestConflict;

// Xc->Xd : capture l'arret physique REEL deja ecoule (StoppedTimer.ET) AU FRONT de
// la nouvelle demande, AVANT le rappel de StoppedTimer plus bas dans ce scan (un TON
// dont IN retombe a FALSE remet son ET a 0 des cet appel — lire apres serait deja 0).
RequestActiveRising(CLK := RequestActive);
IF RequestActiveRising.Q THEN
    CapturedStoppedTime := StoppedTimer.ET;
END_IF;

// Délai plein selon le sens demandé, et base commune pour l'accumulation d'arret
// (le sens final n'est pas encore connu pendant le neutre).
IF ReqAscent AND NOT ReqDescend THEN
    EffectiveDelay := ChangeDelayAscent;
ELSE
    EffectiveDelay := ChangeDelayDescent;
END_IF;
MaxDirectionDelay := MAX(ChangeDelayAscent, ChangeDelayDescent);
// Comparaison AVANT soustraction : TIME est un DWORD non signe cote CODESYS, une
// soustraction dont le resultat mathematique serait negatif (ex: T#500ms - T#800ms)
// deborde silencieusement vers ~T#49j au lieu de saturer a 0 -- MAX(..., T#0ms)
// APRES une soustraction debordee ne corrige rien (le DWORD deborde reste "positif").
IF CapturedStoppedTime >= EffectiveDelay THEN
    RemainingDelay := T#0ms;
ELSE
    RemainingDelay := EffectiveDelay - CapturedStoppedTime;
END_IF;

DirectionChanged := (ReqAscent AND NOT CommandedAscent)
                 OR (ReqDescend AND NOT CommandedDescend)
                 OR (CommandedAscent AND NOT ReqAscent)
                 OR (CommandedDescend AND NOT ReqDescend);

// D18 : au front montant Enable avec sens maintenu, armer le temps mort
// (ne pas re-adopter le sens immediatement — pas de redemarrage inrush).
IF EnableRising AND RequestActive THEN
    DeadTimeArmed := TRUE;
END_IF;

// Xc->Xd : StoppedTimer compte l'arret physique REEL (Enable = treuil arrete,
// contacteurs retombes, cf. FB_Winch) pendant TOUT le neutre, jamais reinitialise
// par le simple relachement du joystick — c'est ce cumul qui alimente la capture
// ci-dessus au scan suivant.
StoppedTimer(IN := Enable AND NOT RequestActive, PT := MaxDirectionDelay);

// Xa->Xb : compte le reliquat (delai plein - arret deja credite) apres la nouvelle
// demande d'inversion.
DirectionChangeDelay(
    IN := Enable AND RequestActive AND DirectionChanged,
    PT := RemainingDelay
);
DelayElapsed := DirectionChangeDelay.ET;

// Adoption du sens
IF NOT RequestActive THEN
    // Neutre ou double demande : aucun sens commandé. Une double demande est
    // explicitement refusée, sans priorité implicite.
    CommandedAscent := FALSE;
    CommandedDescend := FALSE;
    DirectionChangePending := FALSE;
    DeadTimeArmed := FALSE;
ELSIF DirectionChangeDelay.Q THEN
    // Temps mort ecoule : adoption du sens, y compris si DeadTimeArmed etait pose
    // (purge desormais atteignable -- le temps mort minimal a ete respecte, il ne
    // doit pas rester arme indefiniment une fois le delai reellement ecoule).
    CommandedAscent := ReqAscent;
    CommandedDescend := ReqDescend;
    DirectionChangePending := FALSE;
    DeadTimeArmed := FALSE;
ELSIF DeadTimeArmed THEN
    // D18 : temps mort au front Enable — pas d'adoption immediate tant que le
    // delai (ci-dessus) n'est pas ecoule.
    DirectionChangePending := TRUE;
ELSIF NOT (CommandedAscent OR CommandedDescend) THEN
    // Depuis le neutre : depart immediat si reprise du MEME sens (ou premier sens),
    // sinon (sens oppose) pending + delai dedie obligatoire.
    IF (NOT (LastAscent OR LastDescend))
       OR (ReqAscent AND LastAscent)
       OR (ReqDescend AND LastDescend) THEN
        CommandedAscent := ReqAscent;
        CommandedDescend := ReqDescend;
        DirectionChangePending := FALSE;
    ELSE
        DirectionChangePending := TRUE;
    END_IF;
ELSIF DirectionChanged THEN
    // Inversion directe (sans passage au neutre) : pending + delai
    DirectionChangePending := TRUE;
ELSE
    DirectionChangePending := FALSE;
END_IF;

// Memorise le dernier sens non nul ADOPTE (pas la simple demande) : c'est ce sens qui
// sert de reference pour detecter une reprise opposee apres passage au neutre.
IF CommandedAscent OR CommandedDescend THEN
    LastAscent := CommandedAscent;
    LastDescend := CommandedDescend;
END_IF;

// Le sens adopte correspond desormais a la demande (aucune inversion en cours) :
// le credit d'arret est CONSOMME. Une inversion ULTERIEURE sans nouveau passage au
// neutre (RequestActive reste continuellement vrai) ne doit jamais reutiliser un
// arret perime — elle applique alors le delai plein (CapturedStoppedTime := 0).
IF NOT DirectionChangePending AND (CommandedAscent = ReqAscent) AND (CommandedDescend = ReqDescend) THEN
    CapturedStoppedTime := T#0ms;
END_IF;

          
END_FUNCTION_BLOCK

(* ======================================================================= ⚙️ FB_WinchStepShaper — Cadencement de palier (montee cadencee) ─────────────────────────────────────────────────────────────── 🎯 Rôle : Cadence la montee de palier (+1 cran / StepRampDelay), descente immediate a 0 (aucune rampe descendante) 📄 Doc métier : DOC/AF/AF_Partie-10_Fonction_Winch_v2.1.md 🔌 Interface : Brique technique (contrat light, pas de defaut) 🔒 Sécurité : D10 — StepRampDelay dedie, decouple des delais direction ======================================================================= *)
FUNCTION_BLOCK FB_WinchStepShaper
  VAR_INPUT
    Enable : BOOL;  (* --> [CMD] Autorisation FB (TRUE = actif) *)
    TargetStep : INT;  (* --> [CMD] Palier cible demande *)
    StepRampDelay : TIME;  (* --> [CFG] Delai de cadence montee de palier *)
  END_VAR
  VAR_OUTPUT
    ShapedStep : INT;  (* <-- [DIAG] Palier metier temporise actif *)
    StepDelayElapsed : TIME;  (* <-- [DIAG] Ecoule tempo metier palier *)
  END_VAR
  VAR
    StepDelay : TON;  (* . [LOC] Temporisation hausse de palier *)
  END_VAR

            

// === IMPLEMENTATION ===

IF NOT Enable THEN
    ShapedStep := 0;
    StepDelay(IN := FALSE);
    StepDelayElapsed := T#0s;
    RETURN;
END_IF;

// Temporisation : compte quand la cible est au-dessus du palier courant.
// NOT StepDelay.Q : un TON garde .Q TRUE tant que IN est TRUE (pas d'impulsion).
// Sans ce terme, une fois StepRampDelay ecoule le +1 ci-dessous s'appliquerait a
// CHAQUE scan -> montee 1 -> N en quelques scans. Ici le timer se re-arme apres
// chaque cran -> une hausse de palier / StepRampDelay (cascade reelle).
StepDelay(
    IN := (TargetStep > ShapedStep) AND (ShapedStep > 0) AND NOT StepDelay.Q,
    PT := StepRampDelay
);
StepDelayElapsed := StepDelay.ET;

// Cadencement asymetrique : montee +1 cran / StepRampDelay, descente immediate
IF TargetStep = 0 THEN
    ShapedStep := 0;
ELSIF TargetStep < ShapedStep THEN
    ShapedStep := TargetStep;
ELSIF TargetStep > ShapedStep THEN
    IF ShapedStep = 0 THEN
        ShapedStep := 1;
    ELSIF StepDelay.Q THEN
        ShapedStep := ShapedStep + 1;
    END_IF;
END_IF;

          
END_FUNCTION_BLOCK
